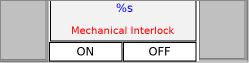
VISUALIZATION Std_OnOffDev_Ctrl  // 249x63
VAR_IN_OUT
	m_Input_Inst : None;
END_VAR
    RoundedRectangle (50,0 146x41), "%s", text variable: m_Input_Inst.IN_DevName
    RoundedRectangle (49,42 73x19), "ON", colour toggle: (m_Input_Inst.S_OnSig) <> 0
    RoundedRectangle (123,42 73x19), "OFF", colour toggle: (NOT m_Input_Inst.S_OnSig) <> 0
    RoundedRectangle (50,21 146x19), "Mechanical Interlock", invisible if: (NOT (NOT m_Input_Inst.In_OnXLock AND m_Input_Inst.T_ManOn)) <> 0
    Group (0,0 46x59)
        tap m_Input_Inst.T_ManOn
        Button (0,0 48x61)
        Polygon (38,51)
        Polygon (35,51)
    Group (199,0 46x59)
        tap m_Input_Inst.T_ManOff
        Button (0,0 48x60)
        Polygon (10,50)
        Polygon (13,50)
END_VISUALIZATION

(* stored: Version 1.1.0.1, ProductVersion 3.1.4018.2
   Visu Std_OnOffDev_Ctrl: Id {526a192b-e8a9-4a22-8599-ed46443b6b7a} *)
